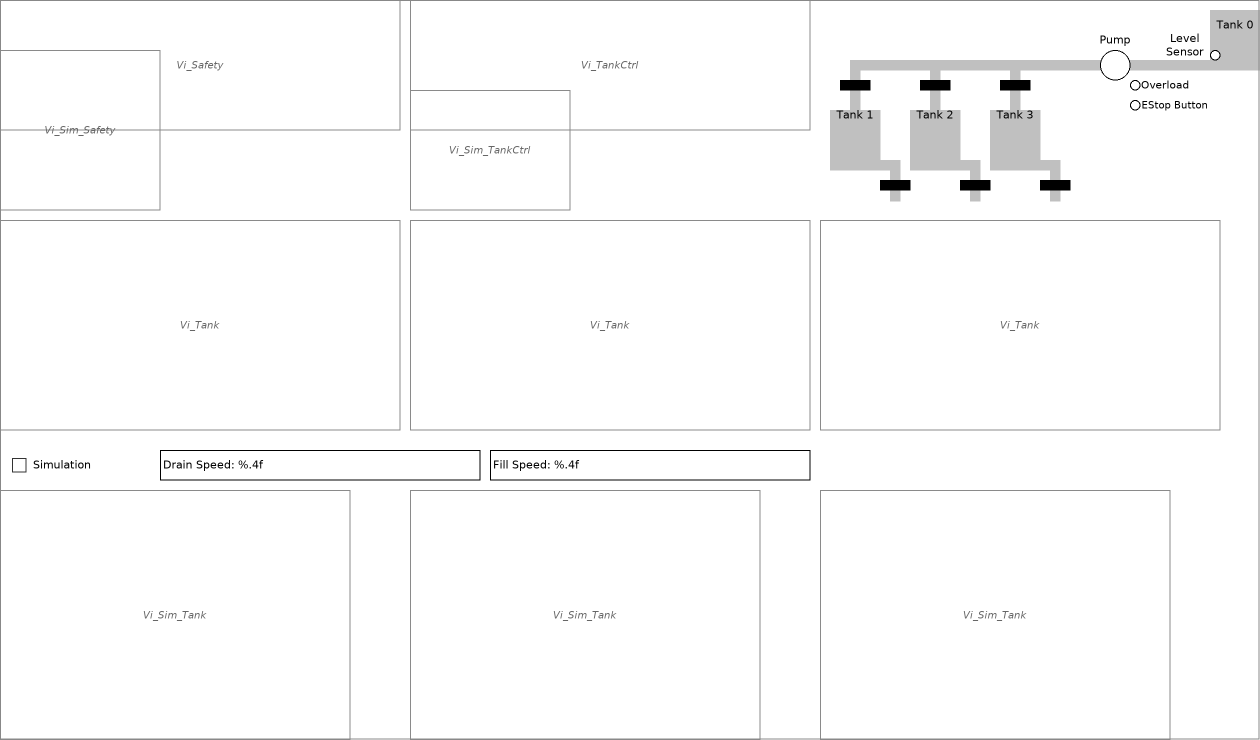
VISUALIZATION MAIN  // 1260x740
    Rectangle (1120,60 140x10)
    Rectangle (1210,10 50x60)
    Frame (0,0 400x130)
        shows Vi_Safety(hmi := MAIN.safety._hmi)
    Frame (0,50 160x160)
        shows Vi_Sim_Safety(obj := MAIN.safety)
    Frame (410,0 400x130)
        shows Vi_TankCtrl(hmi := MAIN.tankCtrl.ctx.hmi)
    Frame (410,90 160x120)
        shows Vi_Sim_TankCtrl(obj := MAIN.tankCtrl)
    Frame (0,220 400x210)
        shows Vi_Tank(hmi := MAIN.tank[1].ctx.hmi)
    Frame (410,220 400x210)
        shows Vi_Tank(hmi := MAIN.tank[2].ctx.hmi)
    Frame (820,220 400x210)
        shows Vi_Tank(hmi := MAIN.tank[3].ctx.hmi)
    Frame (0,490 350x250)
        shows Vi_Sim_Tank(obj := MAIN.tank[1], obj2 := MAIN.outlet[1])
    Frame (410,490 350x250)
        shows Vi_Sim_Tank(obj := MAIN.tank[2], obj2 := MAIN.outlet[2])
    Frame (820,490 350x250)
        shows Vi_Sim_Tank(obj := MAIN.tank[3], obj2 := MAIN.outlet[3])
    Rectangle (850,60 260x10)
    Ellipse (1100,50 30x30), colour toggle: MAIN.tankCtrl.bRunPump
    Rectangle (850,60 10x50)
    Rectangle (930,60 10x50)
    Rectangle (1010,60 10x50)
    Rectangle (970,160 10x41)
    Rectangle (830,110 50x60)
    Rectangle (950,160 30x10)
    Rectangle (910,110 50x60)
    Rectangle (990,110 50x60)
    Rectangle (1050,160 10x41)
    Rectangle (1030,160 30x10)
    Rectangle (890,160 10x41)
    Rectangle (870,160 30x10)
    Ellipse (1210,50 10x10), colour toggle: MAIN.tankCtrl.bNoWater
    Rectangle (1090,30 50x20), "Pump"
    Ellipse (1130,80 10x10), colour toggle: MAIN.tankCtrl.bOverload
    Rectangle (1140,80 50x10), "Overload"
    Rectangle (1160,30 50x30), "Level Sensor"
    Rectangle (1210,10 50x30), "Tank 0"
    Rectangle (990,110 50x10), "Tank 3"
    Rectangle (910,110 50x10), "Tank 2"
    Rectangle (830,110 50x10), "Tank 1"
    Rectangle (1000,80 30x10), invisible if: MAIN.tank[3].bInletValveOpen
    Rectangle (920,80 30x10), invisible if: MAIN.tank[2].bInletValveOpen
    Rectangle (840,80 30x10), invisible if: MAIN.tank[1].bInletValveOpen
    Rectangle (880,180 30x10), invisible if: MAIN.outlet[1].bDrainValveOpen
    Rectangle (960,180 30x10), invisible if: MAIN.outlet[2].bDrainValveOpen
    Rectangle (1040,180 30x10), invisible if: MAIN.outlet[3].bDrainValveOpen
    Ellipse (1130,100 10x10), colour toggle: NOT MAIN.safety.bFeedbackOk
    Rectangle (1140,100 70x10), "EStop Button"
    Checkbox (10,440 140x50), "Simulation", variable: MAIN.sim.bAutoSimEnabled
    Rectangle (160,450 320x30), "Drain Speed: %.4f", text variable: MAIN.sim.fDrainValue.val
        OnMouseUp: write the text variable via Default, min 0
    Rectangle (490,450 320x30), "Fill Speed: %.4f", text variable: MAIN.sim.fFillValue.val
        OnMouseUp: write the text variable via Default, min 0
END_VISUALIZATION

(* stored: Version 1.1.0.1
   Visu MAIN: Id {5260869b-5c1b-4812-baec-e5f9a2a0b333} *)
